// TIA Portal V20 export
// export: Created 2025-12-01T14:56:16.3135335Z, ExportSetting None, DisplayName Totally Integrated Automation Portal, DisplayVersion V20 Update 3, DisplayName TIA Portal Openness, DisplayVersion V20 Update 3, DisplayName TIA Portal Version Control Interface, DisplayVersion V20 Update 3, DisplayName STEP 7 Professional, DisplayVersion V20 Update 3, DisplayName STEP 7 Safety, DisplayVersion V20 Update 2, DisplayName WinCC Basic/Comfort/Advanced, DisplayVersion V20 Update 3, DisplayName WinCC Professional, DisplayVersion V20 Update 3, DisplayName WinCC Unified, DisplayVersion V20 Update 3
TYPE "ROUT_Orden_Fifo_Scanner"
   STRUCT
      Orden : Byte;   // Orden asociada
      Libre : Byte;   // Para adaptar la estructura. Siemens empieza Dints en pares
      Identificador : ULInt;   // CDB
   END_STRUCT;
END_TYPE
